{attribute addProperty BoxType "EL3423-0000-0020"}
{attribute addProperty Id "Total_StatusAT %I*Total_Status_F4CDE3E7144180Total_AdvancedAT %I*Total_Advanced_FCA492E91620Total_Statistic_PowerAT %I*Total_Statistic_Power_A2483F97288360Total_Statistic_PQFAT %I*Total_Statistic_PQF_4F621FA496120Total_Active_ReducedAT %I*Total_Active_Reduced_20E5A44A6480Total_Apparent_ReducedAT %I*Total_Apparent_Reduced_DCF053096480Total_Reactive_ReducedAT %I*Total_Reactive_Reduced_A96F08556480Total_Interval_Energy_ReducedAT %I*Total_Interval_Energy_Reduced_B645E209104130Total_IntervalAT %Q*Total_Interval_ABCD96B2810WcStateAT %I*WcState_98A4DF7520.250InfoDataAT %I*InfoData_BC63D37F80100"}
{attribute addProperty CRC "1856244522"}
{attribute addProperty SizeInBites "930"}
{attribute addProperty SizeInBytes "116.25"}
TYPE EL3423_AE18C60F :
STRUCT
	{attribute addProperty Name "Total_Status"}
	Total_Status : Total_Status_F4CDE3E7;
	{attribute addProperty Name "Total_Advanced"}
	Total_Advanced : Total_Advanced_FCA492E9;
	{attribute addProperty Name "Total_Statistic_Power"}
	Total_Statistic_Power : Total_Statistic_Power_A2483F97;
	{attribute addProperty Name "Total_Statistic_PQF"}
	Total_Statistic_PQF : Total_Statistic_PQF_4F621FA4;
	{attribute addProperty Name "Total_Active_Reduced"}
	Total_Active_Reduced : Total_Active_Reduced_20E5A44A;
	{attribute addProperty Name "Total_Apparent_Reduced"}
	Total_Apparent_Reduced : Total_Apparent_Reduced_DCF05309;
	{attribute addProperty Name "Total_Reactive_Reduced"}
	Total_Reactive_Reduced : Total_Reactive_Reduced_A96F0855;
	{attribute addProperty Name "Total_Interval_Energy_Reduced"}
	Total_Interval_Energy_Reduced : Total_Interval_Energy_Reduced_B645E209;
	{attribute addProperty Name "Total_Interval"}
	Total_Interval : Total_Interval_ABCD96B2;
	{attribute addProperty Name "WcState"}
	WcState : WcState_98A4DF75;
	{attribute addProperty Name "InfoData"}
	InfoData : InfoData_BC63D37F;
END_STRUCT
END_TYPE

(* stored: Version 1.2.0.0, ProductVersion 3.1.4024.9
   DUT EL3423_AE18C60F: Id {000a598d-ca37-45f2-93ed-7f5aaa321376} *)
